FUNCTION_BLOCK FB_Coupling

END_FUNCTION_BLOCK

(* stored: Version 1.1.0.1, ProductVersion 3.1.4024.13
   POU FB_Coupling: Id {80ddf6b9-44b4-4562-b94b-ac30f080db20}, SpecialFunc None *)
